FUNCTION_BLOCK GEN_RDT

VAR_INPUT
	Enable		 : BOOL := TRUE ;
	Min_Time_ms	: TIME := t#1s ; (* min Taktzeit *)
	Max_Time_ms	: TIME := t#1.2s ; (* Max Taktzeit *)
	TP_Q		 : TIME := t#100ms ; (* Zeit Ausgang auf TRUE *)
END_VAR
VAR_OUTPUT
	xQ		 : BOOL ;
END_VAR
VAR
	(* Taktgenerator Simulation *)
	tonRDMTimer	: TON ; (* Zeitbaustein Taktgenerator *)
	tof_xQ		: TOF ; (* Ausschaltverzögerung Taktgenerator *)
	tRDMTime	: TIME ; (* Sollzeit *)
	rRDMTime	: REAL ; (* Zufalswert Timer *)
END_VAR

(*
version 1.1	16 mar. 2008
programmer 	J. Schohaus
tested by		Hugo

RDMT generates a defined pulse with pulse width TP_Q at random times. the random time will be defined with an minimum and maximum time.

*)


(*
FUNCTION_BLOCK RDMTimer
###############################################################################
		 Ersteller / author :		 		 		 		 		 J.Schohaus
		 Datum / date:		 		 		 		 		 		 13.07.2007
###############################################################################
		 Änderungen / Datum / Ersteller :		 		 		 		 		 		 		 		 		 		 		 		 		 		 		 
		 moditication / date / author :		 		 
###############################################################################
		 Verwendete Bibliotheken		 ( * werden im Baustein nicht benötigt )
		 		 		 		 Oscat.lib
###############################################################################
Beschreibung:
*)


tonRDMTimer ( IN:= Enable , PT:= tRDMTime );
tof_xQ ( IN:= tonRDMTimer.Q , PT:= TP_Q );
XQ := tof_xq.Q;
IF tonRDMTimer.Q THEN
		 xQ := TRUE ;
		 rRDMTime := RDM ( last:= rRDMTime ) ;
		 tRDMTime := REAL_TO_TIME ( rRDMTime * DINT_TO_REAL(TIME_TO_DINT( Max_Time_ms - Min_Time_ms ) + TIME_TO_DINT(Min_Time_ms ))) ;
		 tonRDMTimer ( IN:= FALSE );
END_IF;

(* revision history
J. Schohaus	19. nov 2007	rev 1.0
	origial version

hm	16. mar. 2008			rev 1.1
	added type conversion to avoid warnings under codesys 3.0
*)

END_FUNCTION_BLOCK

(* stored: Version 1.1.0.1
   POU GEN_RDT: Id {bedbd061-6205-4823-af0e-523618a5e013}, SpecialFunc None *)
